// TIA Portal V17 export
// export: Created 2025-03-12T14:52:38.6597093Z, ExportSetting WithDefaults, DisplayName Totally Integrated Automation Portal, DisplayVersion V17 Update 8, DisplayName TIA Portal Openness, DisplayVersion V17 Update 8, DisplayName TIA Portal Version Control Interface, DisplayVersion V17, DisplayName SINAMICS Startdrive Advanced, DisplayVersion V17 SP2, DisplayName SINAMICS Startdrive G110M, G120, G120C, G120D, G120P, G115D, DisplayVersion V17 SP2, DisplayName SINAMICS Startdrive G130, G150, S120, S150, SINAMICS MV, S210, DisplayVersion V17 SP2, DisplayName STEP 7 Professional, DisplayVersion V17 Update 8, DisplayName SINUMERIK ONE STEP 7 Toolbox, DisplayVersion V17 Update 12, DisplayName SINUMERIK 840D sl STEP 7 Toolbox, DisplayVersion V17 Update 12, DisplayName STEP 7 Safety, DisplayVersion V17 Update 6, DisplayName WinCC Advanced, DisplayVersion V17 Update 8
TYPE "HOPPER PRESSURE CONTROL"
// stored: IsFailsafeCompliant false
   STRUCT
      FAULTED : Bool;
      "START GENERAL CONDITIONS" : Bool;
      "START GENERAL CONDITIONS HELP" : Bool;
      "START INITIAL CONDITIONS" : Bool;
      "START INITIAL CONDITIONS HELP" : Bool;
      "START MANUAL REQUEST" : Bool;
      "FEEDBACK ON" : Bool;
      "START AUTO REQUEST" : Bool;
      "START GLOBAL REQUEST" : Bool;
      "START COMMAND" : Bool;
      "SYSTEM ON" : Bool;
      "STOP GENERAL CONDITIONS" : Bool;
      "STOP GENERAL CONDITIONS HELP" : Bool;
      "STOP INITIAL CONDITIONS" : Bool;
      "STOP INITIAL CONDITIONS HELP" : Bool;
      "STOP MANUAL REQUEST" : Bool;
      "STOP AUTO REQUEST" : Bool;
      "STOP GLOBAL REQUEST" : Bool;
      "STOP COMMAND" : Bool;
      STOPPED : Bool;
      "FEEDBACK OFF" : Bool;
      "CONTROL DONE" : Bool;
      "SETPOINT PRESSURE" : Real;
      "FEEDBACK PRESSURE" : Real;
      "LIM LO" : Real;
      "LIM HI" : Real;
      "HMI START" : Bool;
      "HMI STOP" : Bool;
      "HMI START CONDITIONS" : Bool;
      "HMI STOP CONDITIONS" : Bool;
      "HMI STARTED" : Bool;
      "HMI STOPPED" : Bool;
      "HMI STARTING" : Bool;
      "HMI STOPPING" : Bool;
      "HMI PRESSURE VALUE" : Real;
      HMI_PRESSURE_INCREMENT : Real;
   END_STRUCT;
END_TYPE
